GLOBALCONSTANTS DefaultPool_PWM12 (* Global constants *)
  PACKAGE Uebungen::const::UT::PWM12;
  VAR_GLOBAL CONSTANT
    DataMask_M1 : UINT := 1000;
    DataMask_PWM1 : UINT := 1001;
    DataMask_PWM2 : UINT := 1002;
    DataMask_PWM3 : UINT := 1003;
    SoftKeyMask_PWM : UINT := 4000;
    SoftKey_Eingaenge : UINT := 5000;
    SoftKey_PWM_1 : UINT := 5001;
    SoftKey_PWM_2 : UINT := 5002;
    SoftKey_PWM_3 : UINT := 5003;
    Label_Btn_ZERO : UINT := 11001;
    Label_Btn_DOWN_FAST : UINT := 11002;
    Label_Btn_DOWN_SLOW : UINT := 11003;
    Label_Btn_UP_SLOW : UINT := 11004;
    Label_Btn_UP_FAST : UINT := 11005;
    Label_Btn_FULL : UINT := 11006;
    Label_Q01 : UINT := 11011;
    InputNumber_PWM_Q01 : UINT := 9000;
    NumberVariable_PWM_Q01 : UINT := 21000;
    Bargraph_PWM_Q01 : UINT := 14000;
    Button_PWM_Q01_ZERO : UINT := 6001;
    Button_PWM_Q01_DOWN_FAST : UINT := 6002;
    Button_PWM_Q01_DOWN_SLOW : UINT := 6003;
    Button_PWM_Q01_UP_SLOW : UINT := 6004;
    Button_PWM_Q01_UP_FAST : UINT := 6005;
    Button_PWM_Q01_FULL : UINT := 6006;
    Label_Q02 : UINT := 11012;
    InputNumber_PWM_Q02 : UINT := 9001;
    NumberVariable_PWM_Q02 : UINT := 21001;
    Bargraph_PWM_Q02 : UINT := 14001;
    Button_PWM_Q02_ZERO : UINT := 6007;
    Button_PWM_Q02_DOWN_FAST : UINT := 6008;
    Button_PWM_Q02_DOWN_SLOW : UINT := 6009;
    Button_PWM_Q02_UP_SLOW : UINT := 6010;
    Button_PWM_Q02_UP_FAST : UINT := 6011;
    Button_PWM_Q02_FULL : UINT := 6012;
    Label_Q03 : UINT := 11013;
    InputNumber_PWM_Q03 : UINT := 9002;
    NumberVariable_PWM_Q03 : UINT := 21002;
    Bargraph_PWM_Q03 : UINT := 14002;
    Button_PWM_Q03_ZERO : UINT := 6013;
    Button_PWM_Q03_DOWN_FAST : UINT := 6014;
    Button_PWM_Q03_DOWN_SLOW : UINT := 6015;
    Button_PWM_Q03_UP_SLOW : UINT := 6016;
    Button_PWM_Q03_UP_FAST : UINT := 6017;
    Button_PWM_Q03_FULL : UINT := 6018;
    Label_Q04 : UINT := 11014;
    InputNumber_PWM_Q04 : UINT := 9003;
    NumberVariable_PWM_Q04 : UINT := 21003;
    Bargraph_PWM_Q04 : UINT := 14003;
    Button_PWM_Q04_ZERO : UINT := 6019;
    Button_PWM_Q04_DOWN_FAST : UINT := 6020;
    Button_PWM_Q04_DOWN_SLOW : UINT := 6021;
    Button_PWM_Q04_UP_SLOW : UINT := 6022;
    Button_PWM_Q04_UP_FAST : UINT := 6023;
    Button_PWM_Q04_FULL : UINT := 6024;
    Label_Q05 : UINT := 11015;
    InputNumber_PWM_Q05 : UINT := 9004;
    NumberVariable_PWM_Q05 : UINT := 21004;
    Bargraph_PWM_Q05 : UINT := 14004;
    Button_PWM_Q05_ZERO : UINT := 6025;
    Button_PWM_Q05_DOWN_FAST : UINT := 6026;
    Button_PWM_Q05_DOWN_SLOW : UINT := 6027;
    Button_PWM_Q05_UP_SLOW : UINT := 6028;
    Button_PWM_Q05_UP_FAST : UINT := 6029;
    Button_PWM_Q05_FULL : UINT := 6030;
    Label_Q06 : UINT := 11016;
    InputNumber_PWM_Q06 : UINT := 9005;
    NumberVariable_PWM_Q06 : UINT := 21005;
    Bargraph_PWM_Q06 : UINT := 14005;
    Button_PWM_Q06_ZERO : UINT := 6031;
    Button_PWM_Q06_DOWN_FAST : UINT := 6032;
    Button_PWM_Q06_DOWN_SLOW : UINT := 6033;
    Button_PWM_Q06_UP_SLOW : UINT := 6034;
    Button_PWM_Q06_UP_FAST : UINT := 6035;
    Button_PWM_Q06_FULL : UINT := 6036;
    Label_Q07 : UINT := 11017;
    InputNumber_PWM_Q07 : UINT := 9006;
    NumberVariable_PWM_Q07 : UINT := 21006;
    Bargraph_PWM_Q07 : UINT := 14006;
    Button_PWM_Q07_ZERO : UINT := 6037;
    Button_PWM_Q07_DOWN_FAST : UINT := 6038;
    Button_PWM_Q07_DOWN_SLOW : UINT := 6039;
    Button_PWM_Q07_UP_SLOW : UINT := 6040;
    Button_PWM_Q07_UP_FAST : UINT := 6041;
    Button_PWM_Q07_FULL : UINT := 6042;
    Label_Q08 : UINT := 11018;
    InputNumber_PWM_Q08 : UINT := 9007;
    NumberVariable_PWM_Q08 : UINT := 21007;
    Bargraph_PWM_Q08 : UINT := 14007;
    Button_PWM_Q08_ZERO : UINT := 6043;
    Button_PWM_Q08_DOWN_FAST : UINT := 6044;
    Button_PWM_Q08_DOWN_SLOW : UINT := 6045;
    Button_PWM_Q08_UP_SLOW : UINT := 6046;
    Button_PWM_Q08_UP_FAST : UINT := 6047;
    Button_PWM_Q08_FULL : UINT := 6048;
    Label_Q09 : UINT := 11019;
    InputNumber_PWM_Q09 : UINT := 9008;
    NumberVariable_PWM_Q09 : UINT := 21008;
    Bargraph_PWM_Q09 : UINT := 14008;
    Button_PWM_Q09_ZERO : UINT := 6049;
    Button_PWM_Q09_DOWN_FAST : UINT := 6050;
    Button_PWM_Q09_DOWN_SLOW : UINT := 6051;
    Button_PWM_Q09_UP_SLOW : UINT := 6052;
    Button_PWM_Q09_UP_FAST : UINT := 6053;
    Button_PWM_Q09_FULL : UINT := 6054;
    Label_Q10 : UINT := 11020;
    InputNumber_PWM_Q10 : UINT := 9009;
    NumberVariable_PWM_Q10 : UINT := 21009;
    Bargraph_PWM_Q10 : UINT := 14009;
    Button_PWM_Q10_ZERO : UINT := 6055;
    Button_PWM_Q10_DOWN_FAST : UINT := 6056;
    Button_PWM_Q10_DOWN_SLOW : UINT := 6057;
    Button_PWM_Q10_UP_SLOW : UINT := 6058;
    Button_PWM_Q10_UP_FAST : UINT := 6059;
    Button_PWM_Q10_FULL : UINT := 6060;
    Label_Q11 : UINT := 11021;
    InputNumber_PWM_Q11 : UINT := 9010;
    NumberVariable_PWM_Q11 : UINT := 21010;
    Bargraph_PWM_Q11 : UINT := 14010;
    Button_PWM_Q11_ZERO : UINT := 6061;
    Button_PWM_Q11_DOWN_FAST : UINT := 6062;
    Button_PWM_Q11_DOWN_SLOW : UINT := 6063;
    Button_PWM_Q11_UP_SLOW : UINT := 6064;
    Button_PWM_Q11_UP_FAST : UINT := 6065;
    Button_PWM_Q11_FULL : UINT := 6066;
    Label_Q12 : UINT := 11022;
    InputNumber_PWM_Q12 : UINT := 9011;
    NumberVariable_PWM_Q12 : UINT := 21011;
    Bargraph_PWM_Q12 : UINT := 14011;
    Button_PWM_Q12_ZERO : UINT := 6067;
    Button_PWM_Q12_DOWN_FAST : UINT := 6068;
    Button_PWM_Q12_DOWN_SLOW : UINT := 6069;
    Button_PWM_Q12_UP_SLOW : UINT := 6070;
    Button_PWM_Q12_UP_FAST : UINT := 6071;
    Button_PWM_Q12_FULL : UINT := 6072;
    Container_I : UINT := 3001;
    Button_I01 : UINT := 6101;
    Button_I02 : UINT := 6102;
    Button_I03 : UINT := 6103;
    Button_I04 : UINT := 6104;
    Button_I05 : UINT := 6105;
    Button_I06 : UINT := 6106;
    Button_I07 : UINT := 6107;
    Button_I08 : UINT := 6108;
    OutputNumber_Tick : UINT := 12020;
    FontAttributes_6x8 : UINT := 23000;
    FontAttributes_24x32 : UINT := 23001;
    Logos_icon : UINT := 20500;
    AuxFunction2_X1 : UINT := 31000;
    WorkingSet : UINT := 0;
  END_VAR
END_GLOBALCONSTANTS
